FUNCTION_BLOCK Calamity_HMI (* Service Interface Function Block Type *)
  (* Standard: 61499-2 *)
  (* Version 0.0, 6/21/2026, Schneider Electric, template *)
  PACKAGE SE.Nereda;
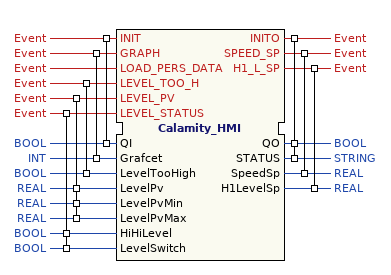
  EVENT_INPUT
    INIT WITH QI;
    GRAPH WITH Grafcet;
    LOAD_PERS_DATA;
    LEVEL_TOO_H WITH LevelTooHigh;
    LEVEL_PV WITH LevelPv, LevelPvMin, LevelPvMax;
    LEVEL_STATUS WITH HiHiLevel, LevelSwitch;
  END_EVENT
  EVENT_OUTPUT
    INITO WITH QO, STATUS;
    SPEED_SP WITH SpeedSp;
    H1_L_SP WITH H1LevelSp;
  END_EVENT
  VAR_INPUT
    QI : BOOL;
    Grafcet : INT;
    LevelTooHigh : BOOL;
    LevelPv : REAL;
    LevelPvMin : REAL;
    LevelPvMax : REAL;
    HiHiLevel : BOOL;
    LevelSwitch : BOOL;
  END_VAR
  VAR_OUTPUT
    QO : BOOL; (* Event Output Qualifier *)
    STATUS : STRING; (* Service Status *)
    SpeedSp : REAL;
    H1LevelSp : REAL;
  END_VAR
  SERVICE /
    SEQUENCE 
    END_SEQUENCE
  END_SERVICE
END_FUNCTION_BLOCK
